PROGRAM MAIN
VAR
END_VAR

END_PROGRAM

(* stored: Version 1.1.0.1
   POU MAIN: Id {5ba26460-ed55-4422-9f9f-678c1b9378de} *)
